// SIMATIC S7-200 project (STEP 7-Micro/WIN), CPU 221 REL 01.10

ORGANIZATION_BLOCK MAIN:OB1
TITLE=
BEGIN
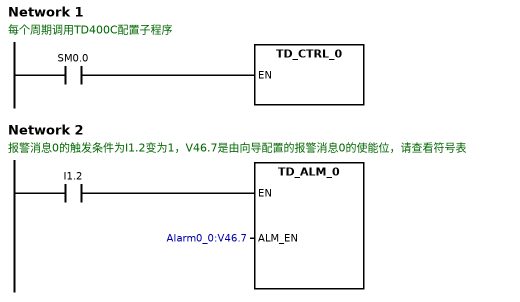
Network 1
// 每个周期调用TD400C配置子程序
LD     SM0.0
CALL   TD_CTRL_0:SBR1
Network 2
// 报警消息0的触发条件为I1.2变为1，V46.7是由向导配置的报警消息0的使能位，请查看符号表
// (network saved uncompiled; LAD cells follow)
// row 0: c0 -| |- I1.2  c1 --  c2 [TD_ALM_0 EN:=power@row0, ALM_EN:=Alarm0_0:V46.7]
// row 1: c2 [box]
END_ORGANIZATION_BLOCK

// SBR1: protected block, not included

// SBR2: protected block, not included

// (further data pages could not be read)
